FUNCTION_BLOCK TestComposite (* Composite FB wrapping other FBs *)
  (* Standard: 61499-2 *)
  (* Version 1.0, 2023-10-04, franz *)
  PACKAGE FBs::Ventilsteuerung;
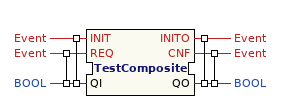
  EVENT_INPUT
    INIT WITH QI; (* Initialization Request *)
    REQ WITH QI; (* Normal Execution Request *)
  END_EVENT
  EVENT_OUTPUT
    INITO WITH QO; (* Initialization Confirm *)
    CNF WITH QO; (* Execution Confirmation *)
  END_EVENT
  VAR_INPUT
    QI : BOOL; (* Input event qualifier *)
  END_VAR
  VAR_OUTPUT
    QO : BOOL; (* Output event qualifier *)
  END_VAR
  EVENT_CONNECTIONS
    INIT TO INITO;
    REQ TO CNF;
  END_CONNECTIONS
  DATA_CONNECTIONS
    QI TO QO;
  END_CONNECTIONS
END_FUNCTION_BLOCK
